PROGRAM FunctionsAndFunctionBlocksex02
VAR
number1 		: number;
number2			: number;
sum12			: number;
END_VAR

number1 * number2 := sum12;

END_PROGRAM

(* stored: Version 1.1.0.1
   POU FunctionsAndFunctionBlocksex02: Id {1e9dea47-b0a3-4534-be8d-089cb81a0bfe}, SpecialFunc None *)
